PROGRAM SiemensControl
VAR
	r_CurrentLimMax						: REAL;
	r_CurrentLimMin						: REAL;
	fbRangeMinSoC : fbValueOutOfRange;
	fbRangeMaxSoC : fbValueOutOfRange;
	fbRangeVoltageDroop : fbValueOutOfRange;
	fbRangeFrequencyDroop : fbValueOutOfRange;
	fbRangeNomVoltage : fbValueOutOfRange;
	fbRangeNomFrequency : fbValueOutOfRange;
	fbRangeCurrentLimMax : fbValueOutOfRange;
	fbRangeCurrentLimMin : fbValueOutOfRange;
	fbRangeBaseCurrentRef : fbValueOutOfRange;
	fbRangeReactCurrentRef : fbValueOutOfRange;
	fbRangeRampRate : fbValueOutOfRange;
	
	w_TypeOfError								: WORD;
	b_TEST										: BOOL;
	
END_VAR

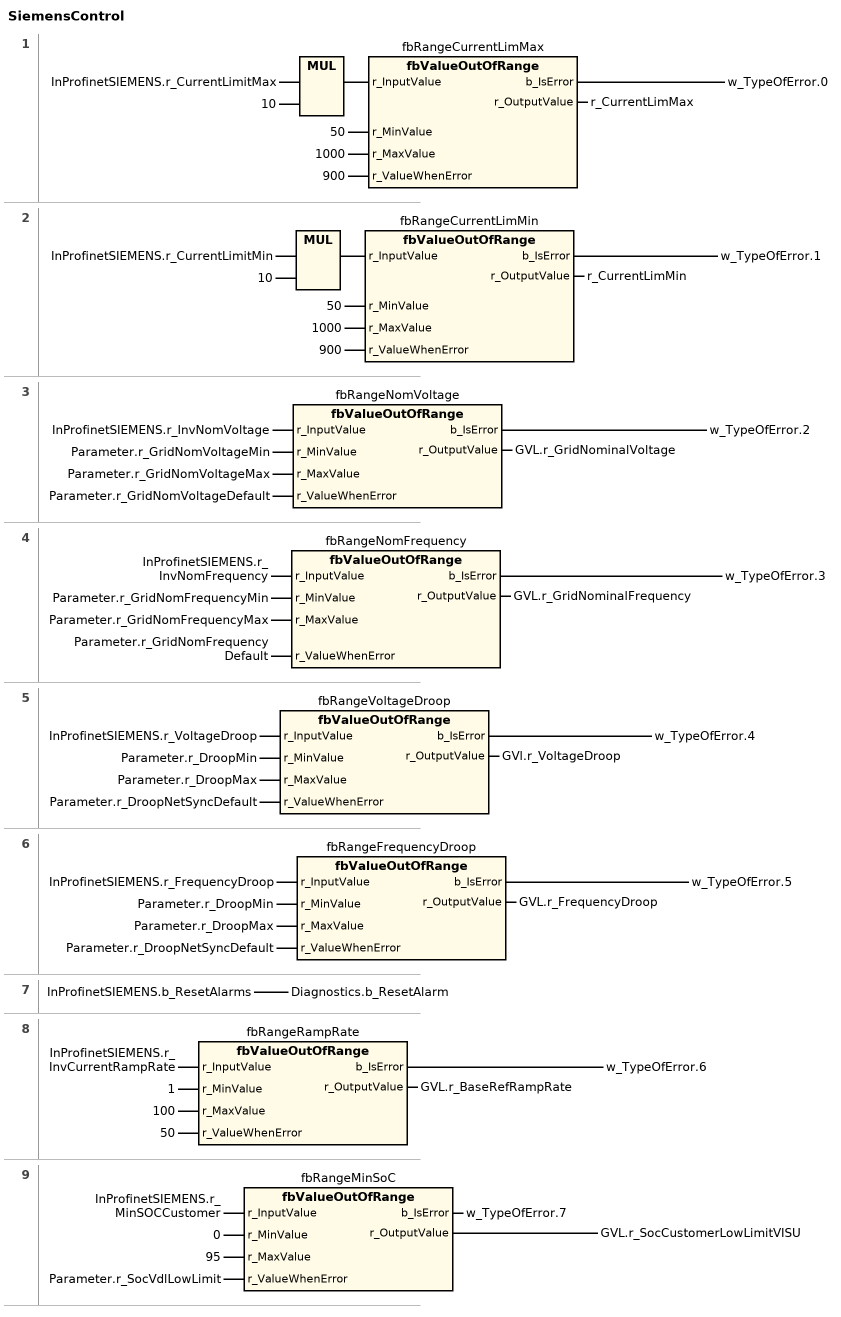
// NETWORK 1
fbRangeCurrentLimMax(
    r_InputValue := InProfinetSIEMENS.r_CurrentLimitMax * 10,
    r_MinValue := 50,
    r_MaxValue := 1000,
    r_ValueWhenError := 900,
    r_OutputValue => r_CurrentLimMax); // fbValueOutOfRange
w_TypeOfError.0 := fbRangeCurrentLimMax.b_IsError;

// NETWORK 2
fbRangeCurrentLimMin(
    r_InputValue := InProfinetSIEMENS.r_CurrentLimitMin * 10,
    r_MinValue := 50,
    r_MaxValue := 1000,
    r_ValueWhenError := 900,
    r_OutputValue => r_CurrentLimMin); // fbValueOutOfRange
w_TypeOfError.1 := fbRangeCurrentLimMin.b_IsError;

// NETWORK 3
fbRangeNomVoltage(
    r_InputValue := InProfinetSIEMENS.r_InvNomVoltage,
    r_MinValue := Parameter.r_GridNomVoltageMin,
    r_MaxValue := Parameter.r_GridNomVoltageMax,
    r_ValueWhenError := Parameter.r_GridNomVoltageDefault,
    r_OutputValue => GVL.r_GridNominalVoltage); // fbValueOutOfRange
w_TypeOfError.2 := fbRangeNomVoltage.b_IsError;

// NETWORK 4
fbRangeNomFrequency(
    r_InputValue := InProfinetSIEMENS.r_InvNomFrequency,
    r_MinValue := Parameter.r_GridNomFrequencyMin,
    r_MaxValue := Parameter.r_GridNomFrequencyMax,
    r_ValueWhenError := Parameter.r_GridNomFrequencyDefault,
    r_OutputValue => GVL.r_GridNominalFrequency); // fbValueOutOfRange
w_TypeOfError.3 := fbRangeNomFrequency.b_IsError;

// NETWORK 5
fbRangeVoltageDroop(
    r_InputValue := InProfinetSIEMENS.r_VoltageDroop,
    r_MinValue := Parameter.r_DroopMin,
    r_MaxValue := Parameter.r_DroopMax,
    r_ValueWhenError := Parameter.r_DroopNetSyncDefault,
    r_OutputValue => GVl.r_VoltageDroop); // fbValueOutOfRange
w_TypeOfError.4 := fbRangeVoltageDroop.b_IsError;

// NETWORK 6
fbRangeFrequencyDroop(
    r_InputValue := InProfinetSIEMENS.r_FrequencyDroop,
    r_MinValue := Parameter.r_DroopMin,
    r_MaxValue := Parameter.r_DroopMax,
    r_ValueWhenError := Parameter.r_DroopNetSyncDefault,
    r_OutputValue => GVL.r_FrequencyDroop); // fbValueOutOfRange
w_TypeOfError.5 := fbRangeFrequencyDroop.b_IsError;

// NETWORK 7
Diagnostics.b_ResetAlarm := InProfinetSIEMENS.b_ResetAlarms;

// NETWORK 8
fbRangeRampRate(
    r_InputValue := InProfinetSIEMENS.r_InvCurrentRampRate,
    r_MinValue := 1,
    r_MaxValue := 100,
    r_ValueWhenError := 50,
    r_OutputValue => GVL.r_BaseRefRampRate); // fbValueOutOfRange
w_TypeOfError.6 := fbRangeRampRate.b_IsError;

// NETWORK 9
fbRangeMinSoC(
    r_InputValue := InProfinetSIEMENS.r_MinSOCCustomer,
    r_MinValue := 0,
    r_MaxValue := 95,
    r_ValueWhenError := Parameter.r_SocVdlLowLimit,
    b_IsError => w_TypeOfError.7); // fbValueOutOfRange
GVL.r_SocCustomerLowLimitVISU := fbRangeMinSoC.r_OutputValue;

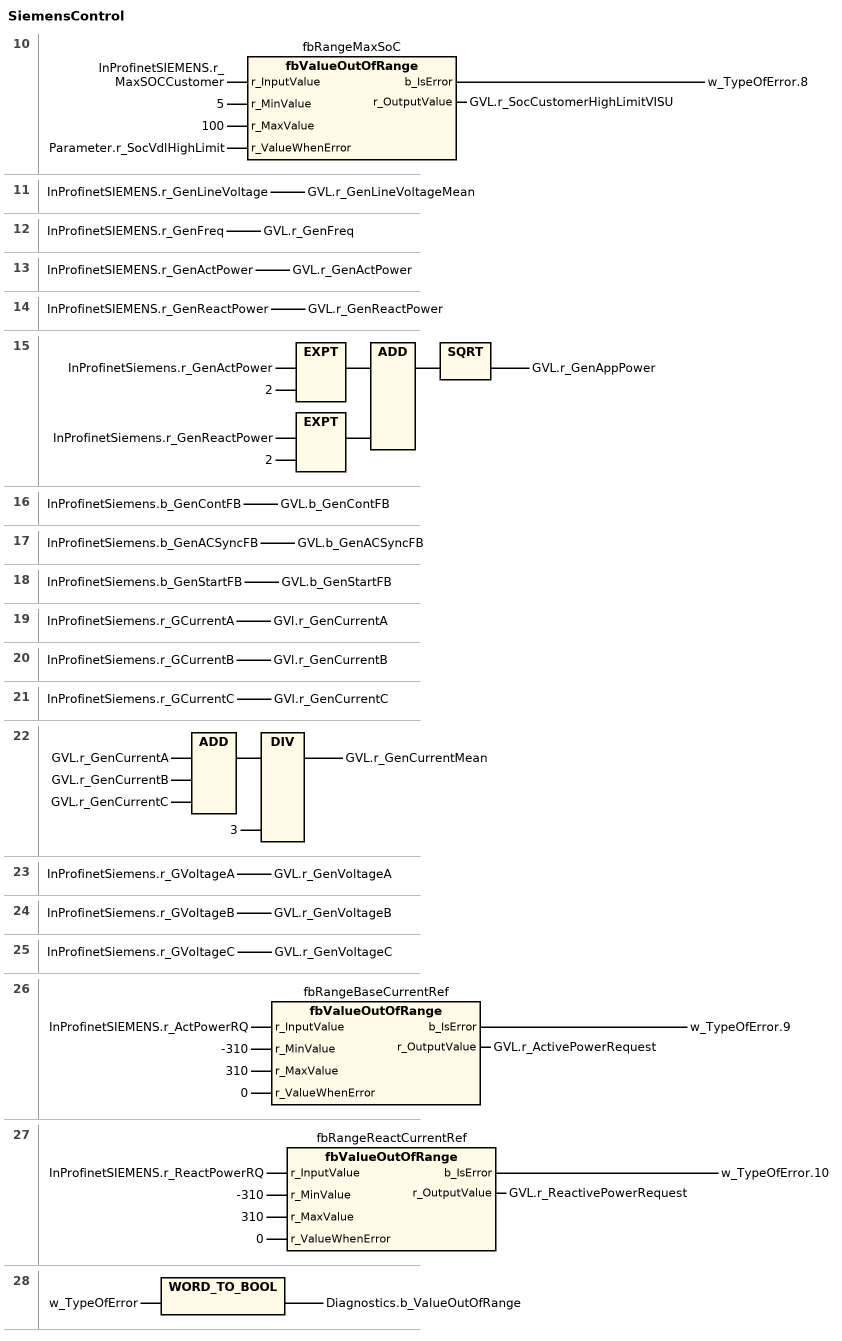
// NETWORK 10
fbRangeMaxSoC(
    r_InputValue := InProfinetSIEMENS.r_MaxSOCCustomer,
    r_MinValue := 5,
    r_MaxValue := 100,
    r_ValueWhenError := Parameter.r_SocVdlHighLimit,
    r_OutputValue => GVL.r_SocCustomerHighLimitVISU); // fbValueOutOfRange
w_TypeOfError.8 := fbRangeMaxSoC.b_IsError;

// NETWORK 11
GVL.r_GenLineVoltageMean := InProfinetSIEMENS.r_GenLineVoltage;

// NETWORK 12
GVL.r_GenFreq := InProfinetSIEMENS.r_GenFreq;

// NETWORK 13
GVL.r_GenActPower := InProfinetSIEMENS.r_GenActPower;

// NETWORK 14
GVL.r_GenReactPower := InProfinetSIEMENS.r_GenReactPower;

// NETWORK 15
GVL.r_GenAppPower := SQRT(EXPT(InProfinetSiemens.r_GenActPower, 2) + EXPT(InProfinetSiemens.r_GenReactPower, 2));

// NETWORK 16
GVL.b_GenContFB := InProfinetSiemens.b_GenContFB;

// NETWORK 17
GVL.b_GenACSyncFB := InProfinetSiemens.b_GenACSyncFB;

// NETWORK 18
GVL.b_GenStartFB := InProfinetSiemens.b_GenStartFB;

// NETWORK 19
GVl.r_GenCurrentA := InProfinetSiemens.r_GCurrentA;

// NETWORK 20
GVl.r_GenCurrentB := InProfinetSiemens.r_GCurrentB;

// NETWORK 21
GVl.r_GenCurrentC := InProfinetSiemens.r_GCurrentC;

// NETWORK 22
GVL.r_GenCurrentMean := (GVL.r_GenCurrentA + GVL.r_GenCurrentB + GVL.r_GenCurrentC) / 3;

// NETWORK 23
GVL.r_GenVoltageA := InProfinetSiemens.r_GVoltageA;

// NETWORK 24
GVL.r_GenVoltageB := InProfinetSiemens.r_GVoltageB;

// NETWORK 25
GVL.r_GenVoltageC := InProfinetSiemens.r_GVoltageC;

// NETWORK 26
fbRangeBaseCurrentRef(
    r_InputValue := InProfinetSIEMENS.r_ActPowerRQ,
    r_MinValue := -310,
    r_MaxValue := 310,
    r_ValueWhenError := 0,
    r_OutputValue => GVL.r_ActivePowerRequest); // fbValueOutOfRange
w_TypeOfError.9 := fbRangeBaseCurrentRef.b_IsError;

// NETWORK 27
fbRangeReactCurrentRef(
    r_InputValue := InProfinetSIEMENS.r_ReactPowerRQ,
    r_MinValue := -310,
    r_MaxValue := 310,
    r_ValueWhenError := 0,
    r_OutputValue => GVL.r_ReactivePowerRequest); // fbValueOutOfRange
w_TypeOfError.10 := fbRangeReactCurrentRef.b_IsError;

// NETWORK 28
Diagnostics.b_ValueOutOfRange := WORD_TO_BOOL(w_TypeOfError);

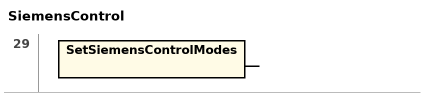
// NETWORK 29
SetSiemensControlModes();

END_PROGRAM

(* stored: Version 1.1.0.1, ProductVersion 3.1.4024.12
   POU SiemensControl: Id {b1931c38-3252-4c34-9009-33198a29a0c7}, SpecialFunc None *)
